// TIA Portal V18 export
FUNCTION "fcCalculVitesse" : Void   // FC5, LAD
// stored: Namespace nsConvoyeur, SetENOAutomatically false
   VAR_INPUT
      ivitesseRPM : UDInt;
   END_VAR
   VAR_OUTPUT
      oVitessePercent : UDInt;
   END_VAR
BEGIN

REGION Network 1
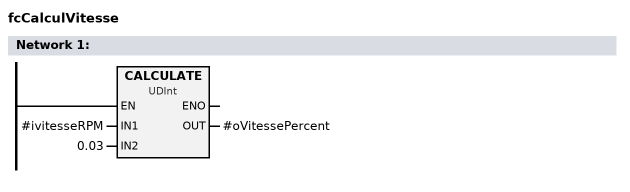
   RUNG wire#powerrail
      { S7_Templates := "SrcType := UDInt"; S7_Expression := "IN1*IN2" } Calculate(in1 := #ivitesseRPM, in2 := 0.03, out => #oVitessePercent)
   END_RUNG
   // the same network as SCL:
   #oVitessePercent := #ivitesseRPM*0.03;
END_REGION
END_FUNCTION
